(* Logix 5000 project; controller ktc_lab10 vendor 1 type 14 code 150 rev 30.11; software revision 30.00 *)

TASK MainTask (continuous, watchdog 500 ms) : MainProgram

MODULES
   Local : vendor 1 type 14 code 150 (Compact 0, rev 30.11)
      Counters : Embedded (Compact 3, rev 1.1, Output RPI 20 ms)
      Discrete_IO : Embedded (Compact 1, rev 3.1, Output RPI 20 ms)
      Analog_IO : Embedded (Compact 2, rev 1.1, Output RPI 80 ms)
END_MODULES

PROGRAM MainProgram   (* main routine MainRoutine *)
VAR
   constant : DINT := 15000;
   current : DINT := 9699;
   PL0 : ALIAS FOR Local:1:O.Data.0;   // LED
   Voltage : DINT := 5473;
   voltage_1 : DINT;
END_VAR

ROUTINE MainRoutine   (* ladder *)
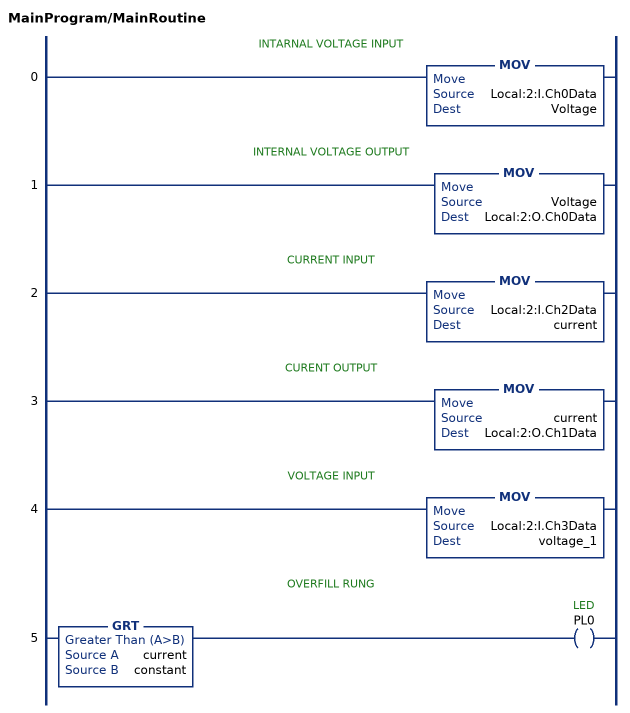
   // INTARNAL VOLTAGE INPUT
   0: MOV(Local:2:I.Ch0Data,Voltage);
   // INTERNAL VOLTAGE OUTPUT
   1: MOV(Voltage,Local:2:O.Ch0Data);
   // CURRENT INPUT
   2: MOV(Local:2:I.Ch2Data,current);
   // CURENT OUTPUT
   3: MOV(current,Local:2:O.Ch1Data);
   // VOLTAGE INPUT
   4: MOV(Local:2:I.Ch3Data,voltage_1);
   // OVERFILL RUNG
   5: GRT(current,constant)OTE(PL0);
END_ROUTINE
END_PROGRAM
